PROGRAM MAIN
VAR
END_VAR

FIS_pgr();

Test_fbFis();

END_PROGRAM

(* stored: Version 1.1.0.1, ProductVersion 3.1.4024.6
   POU MAIN: Id {73f5d705-ee79-4f84-b027-343b752c5397}, SpecialFunc None *)
